FUNCTION_BLOCK FB_CylinderSimul
VAR_INPUT
	moveFwd: BOOL;
	moveBwd: BOOL;
	course:LREAL:=500;	//cylinder course in mm
	moveVel:LREAL:=100;	//move velocity in mm/s
	cycleTime:TIME:=T#10MS;
END_VAR
VAR_OUTPUT
	sensorCylFwd: BOOL;
	sensorCylBwd: BOOL;
	currentPos:LREAL;
	posPercent:LREAL;
END_VAR
VAR
	movementPerCycle: LREAL;
END_VAR

movementPerCycle:= TIME_TO_LREAL(cycletime)/1000*moveVel;
IF moveFwd AND NOT moveBwd THEN
	m_CylFwd();
ELSIF moveBwd AND NOT moveFwd THEN
	m_CylBwd();
END_IF

sensorCylBwd:= currentPos <= 1;
sensorCylFwd:= currentPos >= (course - 1);

METHOD m_CylBwd : BOOL
VAR_INPUT
END_VAR
currentPos:= LIMIT(0,currentPos-movementPerCycle,course);
posPercent:= currentPos*100/course;
END_METHOD

METHOD m_CylFwd : BOOL
VAR_INPUT
END_VAR
currentPos:= LIMIT(0,currentPos+movementPerCycle,course);
posPercent:= currentPos*100/course;
END_METHOD

END_FUNCTION_BLOCK

(* stored: Version 1.1.0.1, ProductVersion 3.1.4024.12
   POU FB_CylinderSimul: Id {86309f97-5da7-417a-87bb-acd077ebc977}, SpecialFunc None
   Method m_CylBwd: Id {0b1130a6-bf15-4c43-ae1d-a2a64047ba68}
   Method m_CylFwd: Id {e0b4e065-4744-4854-9424-04265b2c5d03} *)
